FUNCTION_BLOCK FB_Robot
VAR_INPUT
END_VAR
VAR_OUTPUT
END_VAR
VAR
END_VAR

METHOD RSR1 : BOOL
VAR_INPUT
END_VAR
END_METHOD

METHOD RSR2 : BOOL
VAR_INPUT
END_VAR
END_METHOD

END_FUNCTION_BLOCK

(* stored: Version 1.1.0.1
   POU FB_Robot: Id {0554418f-bec8-43af-97bb-406df361b39b}, SpecialFunc None
   Method RSR1: Id {48966531-33d7-40db-9302-bba9452c9bd2}
   Method RSR2: Id {ac5a31e9-fda5-4a1f-a31a-def60ce2e6e5} *)
